TYPE DriveOutputs :
STRUCT
	SetCounterValue : UDINT;
	TargetPosition : UDINT;
	TargetVelocity : INT;
	StartType : UINT;
	TargetAcceleration : UINT;
	TargetDeceleration : UINT;
END_STRUCT
END_TYPE

(* stored: Version 1.1.0.1, ProductVersion 3.1.4024.9
   DUT DriveOutputs: Id {9202663e-1907-40a8-b3ca-b54202f5f983} *)
